TYPE ST_BusTaster6F_Output :
STRUCT
	bButtons    :ARRAY[1..6] OF BOOL;       (*aktueller Tasterstatus (TRUE = gedrückt)*)
	bButtonsExt :ARRAY[1..6] OF BOOL;       (*aktueller Tasterstatus (TRUE = gedrückt)*)
	
	lrTemp		:LREAL;						(* Temperatur Sensor	*)
	lrRhd		:LREAL;						(* Luftfeuchtigkeit Sensor	*)
	lrBrs		:LREAL;						(* Helligkeit Sensor *)
	
	bCOM			:BOOL;					(*Zeigt die Kommunikation an *)
	bStartupDone	:BOOL;
	
	iState			:BOOL;
	sState			:STRING;
	bError			:BOOL;
	
	tLastUpdateTemp	:TIME;					(* Zeit- Letztes Update Temperatur *)
	tLastUpdateRhd	:TIME;					(* Zeit- Letztes Update Luftfeuchte *)
	tLastUpdateBrs	:TIME;					(* Zeit- Letztes Update Helligkeit *)
	
	sLastUpdateTemp	:STRING(12);			(* Zeit- Letztes Update Temperatur Uhrzeit *)
	sLastUpdateRhd	:STRING(12);			(* Zeit- Letztes Update Luftfeuchte Uhrzeit*)
	sLastUpdateBrs	:STRING(12);			(* Zeit- Letztes Update Helligkeit Uhrzeit*)
	
	dwChanges		:DWORD;					(* Änderungszähler für Startups *)
END_STRUCT
END_TYPE

(* stored: Version 1.1.0.1, ProductVersion 3.1.4024.12
   DUT ST_BusTaster6F_Output: Id {721ad8c1-5593-4dc7-9556-41d037615b47} *)
